// TIA Portal V18 export
// export: Created 2026-06-12T02:00:00Z, ExportSetting WithDefaults, DisplayName Totally Integrated Automation Portal, DisplayVersion V18, DisplayName TIA Portal Openness, DisplayVersion V18
TagTable "AI_B3_Tags"
  AI_B3_Sequence_Count : Real  (PLC tag AI_B3_Sequence_Count, HMI_Connection_1, 1 s)   // COUNT 0-100
  AI_B3_Flow_CIP_Center : Real  (PLC tag AI_B3_Flow_CIP_Center, HMI_Connection_1, 1 s)   // FLOW 100-200 L/h
  AI_B3_Temp_CIP_Upper : Real  (PLC tag AI_B3_Temp_CIP_Upper, HMI_Connection_1, 1 s)   // TEMP 50-80 °C
  AI_B3_Pressure_CIP_1 : Real  (PLC tag AI_B3_Pressure_CIP_1, HMI_Connection_1, 1 s)   // PRESSURE 7-8 bar
  AI_B3_Temp_Chaff_1 : Real  (PLC tag AI_B3_Temp_Chaff_1, HMI_Connection_1, 1 s)   // TEMP 50-80 °C
  AI_B3_Flow_CIP_Feed : Real  (PLC tag AI_B3_Flow_CIP_Feed, HMI_Connection_1, 1 s)   // FLOW 100-200 L/h
  AI_B3_Temp_Steam_1 : Real  (PLC tag AI_B3_Temp_Steam_1, HMI_Connection_1, 1 s)   // TEMP 50-80 °C
  AI_B3_Flow_UCWW_1 : Real  (PLC tag AI_B3_Flow_UCWW_1, HMI_Connection_1, 1 s)   // FLOW 100-200 L/h
  AI_B3_RPM_Screw_Conv : Real  (PLC tag AI_B3_RPM_Screw_Conv, HMI_Connection_1, 1 s)   // RPM 800-1200 RPM
  AI_B3_Temp_Condensate_1 : Real  (PLC tag AI_B3_Temp_Condensate_1, HMI_Connection_1, 1 s)   // TEMP 50-80 °C
  AI_B3_Pressure_Screw_1 : Real  (PLC tag AI_B3_Pressure_Screw_1, HMI_Connection_1, 1 s)   // PRESSURE 7-8 bar
  AI_B3_Flow_CWW_Out : Real  (PLC tag AI_B3_Flow_CWW_Out, HMI_Connection_1, 1 s)   // FLOW 100-200 L/h
  AI_B3_Pressure_CWW_1 : Real  (PLC tag AI_B3_Pressure_CWW_1, HMI_Connection_1, 1 s)   // PRESSURE 7-8 bar
  AI_B3_Temp_Decanter2 : Real  (PLC tag AI_B3_Temp_Decanter2, HMI_Connection_1, 1 s)   // TEMP 50-80 °C
  AI_B3_RPM_Rotary2 : Real  (PLC tag AI_B3_RPM_Rotary2, HMI_Connection_1, 1 s)   // RPM 800-1200 RPM
  AI_B3_RPM_Rotary1 : Real  (PLC tag AI_B3_RPM_Rotary1, HMI_Connection_1, 1 s)   // RPM 800-1200 RPM
  AI_B3_Temp_GroundSilo : Real  (PLC tag AI_B3_Temp_GroundSilo, HMI_Connection_1, 1 s)   // TEMP 50-80 °C
  AI_B3_Flow_GroundSilo : Real  (PLC tag AI_B3_Flow_GroundSilo, HMI_Connection_1, 1 s)   // FLOW 100-200 L/h
  AI_B3_Pressure_Mid_1 : Real  (PLC tag AI_B3_Pressure_Mid_1, HMI_Connection_1, 1 s)   // PRESSURE 7-8 bar
  AI_B3_Flow_Condensate : Real  (PLC tag AI_B3_Flow_Condensate, HMI_Connection_1, 1 s)   // FLOW 100-200 L/h
  AI_B3_Flow_Sump_Out : Real  (PLC tag AI_B3_Flow_Sump_Out, HMI_Connection_1, 1 s)   // FLOW 100-200 L/h
  AI_B3_Level_Sump : Real  (PLC tag AI_B3_Level_Sump, HMI_Connection_1, 1 s)   // LEVEL 30-80 %
  AI_B3_Pressure_Decant1 : Real  (PLC tag AI_B3_Pressure_Decant1, HMI_Connection_1, 1 s)   // PRESSURE 7-8 bar
  AI_B3_Pressure_Decant2 : Real  (PLC tag AI_B3_Pressure_Decant2, HMI_Connection_1, 1 s)   // PRESSURE 7-8 bar
  AI_B3_Flow_Decant1 : Real  (PLC tag AI_B3_Flow_Decant1, HMI_Connection_1, 1 s)   // FLOW 100-200 L/h
  AI_B3_Temp_Decant1 : Real  (PLC tag AI_B3_Temp_Decant1, HMI_Connection_1, 1 s)   // TEMP 50-80 °C
  AI_B3_Temp_FBB_Boiler : Real  (PLC tag AI_B3_Temp_FBB_Boiler, HMI_Connection_1, 1 s)   // TEMP 50-80 °C
  AI_B3_Temp_CWW_Out : Real  (PLC tag AI_B3_Temp_CWW_Out, HMI_Connection_1, 1 s)   // TEMP 50-80 °C
  AI_B3_Pressure_SUMP : Real  (PLC tag AI_B3_Pressure_SUMP, HMI_Connection_1, 1 s)   // PRESSURE 7-8 bar
  AI_B3_Flow_SUMP : Real  (PLC tag AI_B3_Flow_SUMP, HMI_Connection_1, 1 s)   // FLOW 100-200 L/h
  AI_B3_Level_CWW : Real  (PLC tag AI_B3_Level_CWW, HMI_Connection_1, 1 s)   // LEVEL 30-80 %
  AI_B3_Temp_FBB_Out : Real  (PLC tag AI_B3_Temp_FBB_Out, HMI_Connection_1, 1 s)   // TEMP 50-80 °C
  AI_B3_Pressure_FBB_Out : Real  (PLC tag AI_B3_Pressure_FBB_Out, HMI_Connection_1, 1 s)   // PRESSURE 7-8 bar
  AI_B3_Flow_FBB_Out : Real  (PLC tag AI_B3_Flow_FBB_Out, HMI_Connection_1, 1 s)   // FLOW 100-200 L/h
